TYPE union_STATE_MON :
UNION
	byState		: BYTE;
	eState		: enum_FB_MON;
END_UNION
END_TYPE

(* stored: Version 1.1.0.1
   DUT union_STATE_MON: Id {263554dd-feae-4afb-8235-60235a23a9b4} *)
